{attribute 'qualified_only'}
{attribute 'strict'}
TYPE E_SafeSequenceState :
(
	IDLE := 0,
	RUNNING := 1,
	FAULT := 2,
	RESET_PENDING := 3
);
END_TYPE

(* stored: Version 1.1.0.1, ProductVersion 3.1.4024.16
   DUT E_SafeSequenceState: Id {bc5a4e50-470e-42ff-b85e-9c7df2d776b8} *)
